FUNCTION_BLOCK FB_PU_Schuetz_Ablaufsteuerung
VAR_IN_OUT
	Zustand			: ST_PU_Schuetz_Zustand;
	Stellwert			: ST_PU_Schuetz_Stellwert;
END_VAR
VAR_INPUT
	Steuerung		: ST_PU_Schuetz_Steuerung;
	Parameter		: ST_PU_Schuetz_Parameter;
END_VAR
VAR_OUTPUT
END_VAR
VAR
	Timer		: TON;
END_VAR

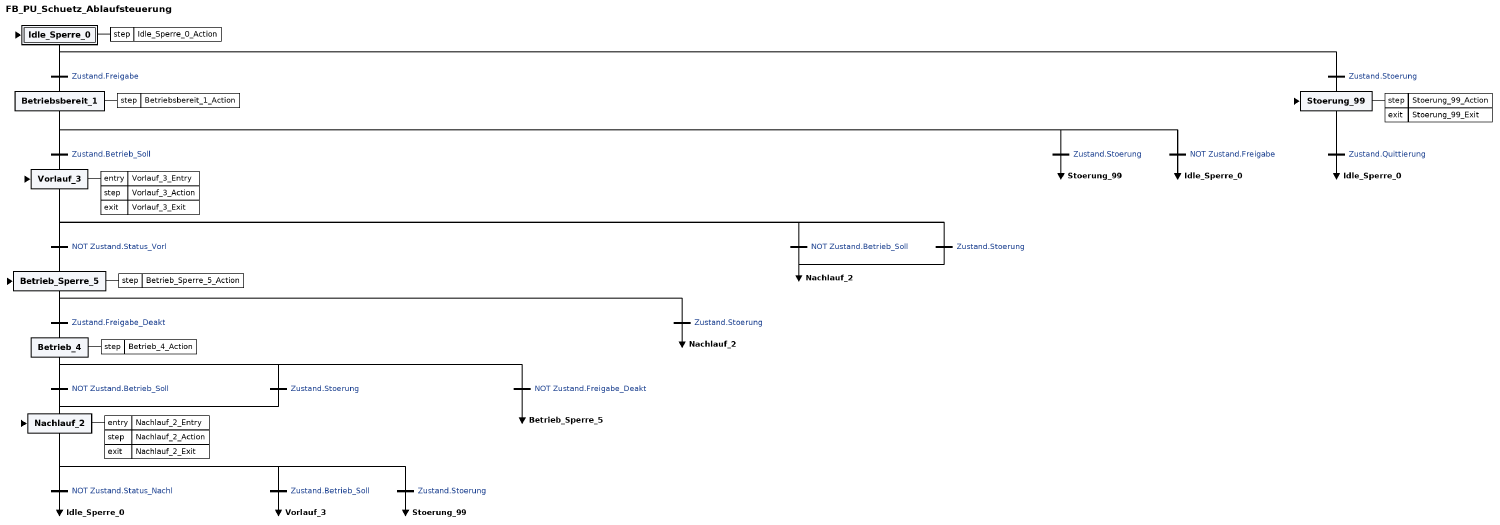
INITIAL_STEP Idle_Sperre_0:
    Idle_Sperre_0_Action(N);  // step action
END_STEP
TRANSITION FROM Idle_Sperre_0 TO Betriebsbereit_1
    := Zustand.Freigabe;
END_TRANSITION
TRANSITION FROM Idle_Sperre_0 TO Stoerung_99
    := Zustand.Stoerung;
END_TRANSITION
STEP Stoerung_99:
    Stoerung_99_Action(N);  // step action
    Stoerung_99_Exit(P0);  // exit action
END_STEP
TRANSITION FROM Stoerung_99 TO Idle_Sperre_0
    := Zustand.Quittierung;
END_TRANSITION
STEP Betriebsbereit_1:
    Betriebsbereit_1_Action(N);  // step action
END_STEP
TRANSITION FROM Betriebsbereit_1 TO Vorlauf_3
    := Zustand.Betrieb_Soll;
END_TRANSITION
TRANSITION FROM Betriebsbereit_1 TO Stoerung_99
    := Zustand.Stoerung;
END_TRANSITION
TRANSITION FROM Betriebsbereit_1 TO Idle_Sperre_0
    := NOT Zustand.Freigabe;
END_TRANSITION
STEP Vorlauf_3:
    Vorlauf_3_Entry(P1);  // entry action
    Vorlauf_3_Action(N);  // step action
    Vorlauf_3_Exit(P0);  // exit action
END_STEP
TRANSITION FROM Vorlauf_3 TO Betrieb_Sperre_5
    := NOT Zustand.Status_Vorl;
END_TRANSITION
TRANSITION FROM Vorlauf_3 TO Nachlauf_2
    := NOT Zustand.Betrieb_Soll;
END_TRANSITION
TRANSITION FROM Vorlauf_3 TO Nachlauf_2
    := Zustand.Stoerung;
END_TRANSITION
STEP Betrieb_Sperre_5:
    Betrieb_Sperre_5_Action(N);  // step action
END_STEP
TRANSITION FROM Betrieb_Sperre_5 TO Betrieb_4
    := Zustand.Freigabe_Deakt;
END_TRANSITION
TRANSITION FROM Betrieb_Sperre_5 TO Nachlauf_2
    := Zustand.Stoerung;
END_TRANSITION
STEP Betrieb_4:
    Betrieb_4_Action(N);  // step action
END_STEP
TRANSITION FROM Betrieb_4 TO Nachlauf_2
    := NOT Zustand.Betrieb_Soll;
END_TRANSITION
TRANSITION FROM Betrieb_4 TO Nachlauf_2
    := Zustand.Stoerung;
END_TRANSITION
TRANSITION FROM Betrieb_4 TO Betrieb_Sperre_5
    := NOT Zustand.Freigabe_Deakt;
END_TRANSITION
STEP Nachlauf_2:
    Nachlauf_2_Entry(P1);  // entry action
    Nachlauf_2_Action(N);  // step action
    Nachlauf_2_Exit(P0);  // exit action
END_STEP
TRANSITION FROM Nachlauf_2 TO Idle_Sperre_0
    := NOT Zustand.Status_Nachl;
END_TRANSITION
TRANSITION FROM Nachlauf_2 TO Vorlauf_3
    := Zustand.Betrieb_Soll;
END_TRANSITION
TRANSITION FROM Nachlauf_2 TO Stoerung_99
    := Zustand.Stoerung;
END_TRANSITION

ACTION Betrieb_4_Action:
(* Stellwert setzen *)
Stellwert.Betrieb := TRUE;
Zustand.Betrieb := Stellwert.Betrieb;

(* Zustand setzen *)
Zustand.Status := E_PU_Zustand_Status_Betrieb;
END_ACTION

ACTION Betrieb_Sperre_5_Action:
(* Stellwert setzen *)
Stellwert.Betrieb := TRUE;

(* Zustand setzen *)
Zustand.Status := E_PU_Zustand_Status_Betrieb_Sperre;
END_ACTION

ACTION Betriebsbereit_1_Action:
(* Stellwert setzen *)
Stellwert.Betrieb := FALSE;

(* Zustand setzen *)
Zustand.Status := E_PU_Zustand_Status_Betriebsbereit;
END_ACTION

ACTION Idle_Sperre_0_Action:
(* Stellwert setzen *)
Stellwert.Betrieb := FALSE;

(* Zustand setzen *)
Zustand.Status := E_PU_Zustand_Status_Idle_Sperre;
END_ACTION

ACTION Nachlauf_2_Action:
(* Nachlauf Timer starten *)
Timer( 	IN := Zustand.Status_Nachl,
		PT := DINT_TO_TIME(Parameter.Zeit_Nachl),
);
Zustand.Status_Nachl	:= NOT Timer.Q;

(* Stellwert setzen *)
Stellwert.Betrieb := FALSE;
Zustand.Betrieb := Stellwert.Betrieb;

(* Zustand setzen *)
Zustand.Status := E_PU_Zustand_Status_Nachl;
END_ACTION

ACTION Nachlauf_2_Entry:
(* Reset Timer *)
Timer(IN := FALSE);
Zustand.Status_Nachl := TRUE;
END_ACTION

ACTION Nachlauf_2_Exit:
Zustand.Status_Nachl := FALSE;
END_ACTION

ACTION Stoerung_99_Action:
(* Stellwert setzen *)
Stellwert.Betrieb := FALSE;

(* Zustand setzen *)
Zustand.Stoerung := TRUE;
Zustand.Status := E_PU_Zustand_Status_Stoerung;
END_ACTION

ACTION Stoerung_99_Exit:
Zustand.Stoerung	:= FALSE;
END_ACTION

ACTION Vorlauf_3_Action:
(* Vorlaufzeit Timer starten *)
Timer( 	IN := Zustand.Status_Vorl,
		PT := DINT_TO_TIME(Parameter.Zeit_Vorl),
);
Zustand.Status_Vorl	:= NOT Timer.Q;

(* Stellwert setzen *)
Stellwert.Betrieb := TRUE;

(* Zustand setzen *)
Zustand.Status := E_PU_Zustand_Status_Vorl;
END_ACTION

ACTION Vorlauf_3_Entry:
(* Reset Timer *)
Timer(IN := FALSE);
Zustand.Status_Vorl := TRUE;
END_ACTION

ACTION Vorlauf_3_Exit:
Zustand.Status_Vorl := FALSE;
END_ACTION

END_FUNCTION_BLOCK

(* stored: Version 1.1.0.1, ProductVersion 3.1.4024.9
   POU FB_PU_Schuetz_Ablaufsteuerung: Id {55055a7e-44a7-4493-ad4d-5153fa92d32c}, SpecialFunc None
   Action Betrieb_4_Action: Id {0d523e0e-7172-4889-84ae-c042a4d7b0b0}
   Action Betrieb_Sperre_5_Action: Id {f63d7b1b-3e99-4009-9660-a7b11f75f328}
   Action Betriebsbereit_1_Action: Id {d522d635-5acf-4470-b850-cdc937bda3d4}
   Action Idle_Sperre_0_Action: Id {50c5396d-2aa4-457a-bcc7-2d71b5e16ab0}
   Action Nachlauf_2_Action: Id {91071e2c-635a-4bb3-ad87-0199a9e88110}
   Action Nachlauf_2_Entry: Id {3601388c-2b53-4313-88d3-ff817ef6026a}
   Action Nachlauf_2_Exit: Id {154f86ce-0263-49a7-a128-f70ff327036f}
   Action Stoerung_99_Action: Id {101b26f3-d156-4994-9744-94295bc884a1}
   Action Stoerung_99_Exit: Id {75eebb95-dbbb-46d5-afea-18d32434e841}
   Action Vorlauf_3_Action: Id {d307c428-87de-43a3-a485-6e5c96020630}
   Action Vorlauf_3_Entry: Id {5d98bb4d-7739-48f2-ba2b-2be0121914bb}
   Action Vorlauf_3_Exit: Id {96aebd28-0ad5-4fda-a149-148fa683275b} *)
